// SIMATIC S7-200 project (STEP 7-Micro/WIN), CPU 221 REL 01.10

SYMBOL_TABLE USER1
MT               I0.0     // mo thuan
MN               I0.1     // mo nguoc
DC_quay_thuan    Q0.0     // dong co quay thuan
DC_quay_nguoc    Q0.1     // dong co quay nguoc
estop            I0.2     // dung
END_SYMBOL_TABLE

ORGANIZATION_BLOCK MAIN:OB1
TITLE=PROGRAM COMMENTS
BEGIN
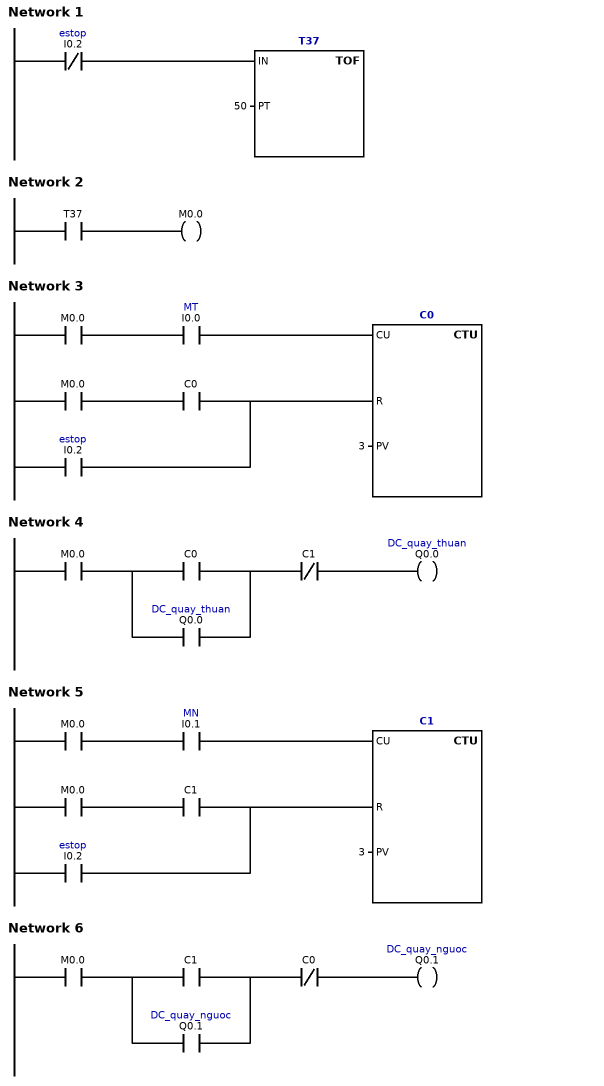
Network 1
LDN    estop:I0.2
TOF    T37, 50
Network 2
LD     T37
=      M0.0
Network 3
LD     M0.0
A      MT:I0.0
LD     M0.0
A      C0
O      estop:I0.2
CTU    C0, 3
Network 4
LD     M0.0
LD     C0
O      DC_quay_thuan:Q0.0
ALD
AN     C1
=      DC_quay_thuan:Q0.0
Network 5
LD     M0.0
A      MN:I0.1
LD     M0.0
A      C1
O      estop:I0.2
CTU    C1, 3
Network 6
LD     M0.0
LD     C1
O      DC_quay_nguoc:Q0.1
ALD
AN     C0
=      DC_quay_nguoc:Q0.1
END_ORGANIZATION_BLOCK
